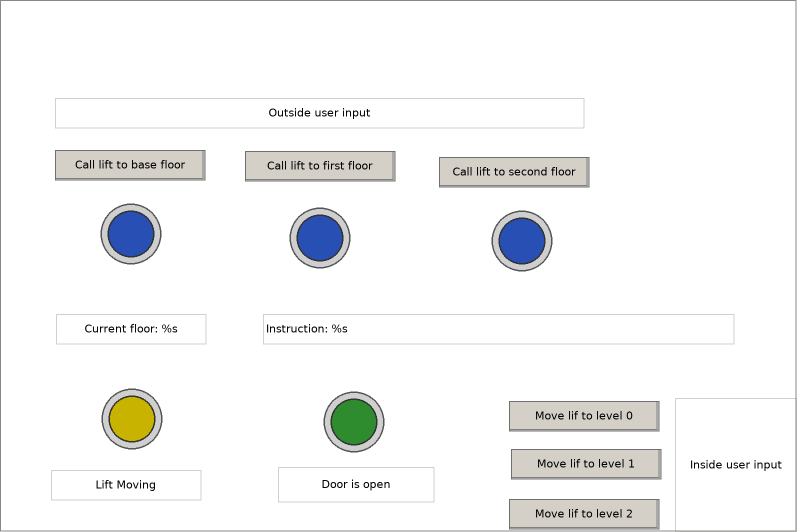
VISUALIZATION Visualization  // 797x532
    Button (55,150 150x30), "Call lift to base floor"
        tap GVL.callLevel0
    Lamp1 (96,199 70x70), variable: ledLogic.ledLevel0, style: Lamp-Lamp1-Blue
    Lamp1 (319,387 70x70), variable: ledLogic.ledDoorsOpen, style: Lamp-Lamp1-Green
    Textfield (51,470 150x30), "Lift Moving"
    Button (245,151 150x30), "Call lift to first floor"
        tap GVL.callLevel1
    Lamp1 (285,203 70x70), variable: ledLogic.ledLevel1, style: Lamp-Lamp1-Blue
    Lamp1 (487,206 70x70), variable: ledLogic.ledLevel2, style: Lamp-Lamp1-Blue
    Button (509,401 150x30), "Move lif to level 0"
        tap GVL.setTargetLevel0
    Lamp1 (97,384 70x70), tooltip "Lift moving", variable: ledLogic.ledLiftMoving, style: Lamp-Lamp1-Yellow
    Textfield (278,467 156x35), "Door is open"
    Button (439,157 150x30), "Call lift to second floor"
        tap GVL.callLevel2
    Button (511,449 150x30), "Move lif to level 1"
        tap GVL.setTargetLevel1
    Button (509,499 150x30), "Move lif to level 2"
        tap GVL.setTargetLevel2
    Textfield (56,314 150x30), "Current floor: %s", text variable: GVL.currentFloor
        p4168582468: GVL.currentFloor
    Textfield (263,314 471x30), "Instruction: %s", text variable: GVL.instructionString
        p4168582468: GVL.currentFloor
    Textfield (55,98 529x30), "Outside user input", text variable: GVL.currentFloor
        p4168582468: GVL.currentFloor
    Textfield (675,398 122x134), "Inside user input"
END_VISUALIZATION

(* stored: Version 1.1.0.1, ProductVersion 3.1.4024.12
   Visu Visualization: Id {5b713095-f953-4139-8fb5-5ac9ac4ded7a} *)
